TYPE E_CommandProcessState :
(
	eNone:=0,
	eDone,
	eProcessing,
	eFail:=-1
);
END_TYPE

(* stored: Version 1.1.0.1, ProductVersion 3.1.0.23
   DUT E_CommandProcessState: Id {9b6fa264-53cd-49e0-a707-95faac547243} *)
